# EPICS autosave request: ADApp/Db/NDROIStatN_settings.req
# This works for one ROI
$(P)$(R)Name
$(P)$(R)Use
$(P)$(R)BgdWidth
$(P)$(R)MinX
$(P)$(R)MinY
$(P)$(R)SizeX
$(P)$(R)SizeY
